FUNCTION_BLOCK FB_Auto_Combination
VAR_INPUT
	bEnable					: BOOL;
END_VAR
VAR_OUTPUT
	fPCV					: LREAL;
	fSCV					: LREAL;
END_VAR
VAR

//Sine Wave
fbClock						: FB_Clock;	
fSineRef					: LREAL;

//Off
fPCV_Off					: LREAL;
fSCV_Off					: LREAL;


//////Primary Control////////
fSCV_On						: LREAL;
fPCV_PC						: LREAL;
	
fbAutoSineMotion_PC			: FB_AutoSineMotion;

/////Secondary Control/////
fPCV_set					: LREAL := 1.0;
fPCV_On						: LREAL;
fSCV_SC						: LREAL;

fbGain_Chooser_P			: FB_GainChooser;
fbGain_Chooser_I			: FB_GainChooser;
fbDerivator					: FB_Derivator;

fbPID_OL					: FB_PID_Controller;
fbDeadband_sine				: FB_Deadband_Auto_sine;
fbDisplacementControl_IL	: FB_DisplacementControl_SC;



//Plotting
fVelref_sine				: LREAL;
fOutPutSignal_OL_combi		: LREAL;
fDeadbandComp_out			: LREAL;

//MUX
fbMUX_selector				: FB_MUX_selector;

END_VAR
VAR // added by the converter: edge detectors and wires of the graphical bodies
    _w1 : LREAL;
    _w2 : BOOL;
END_VAR

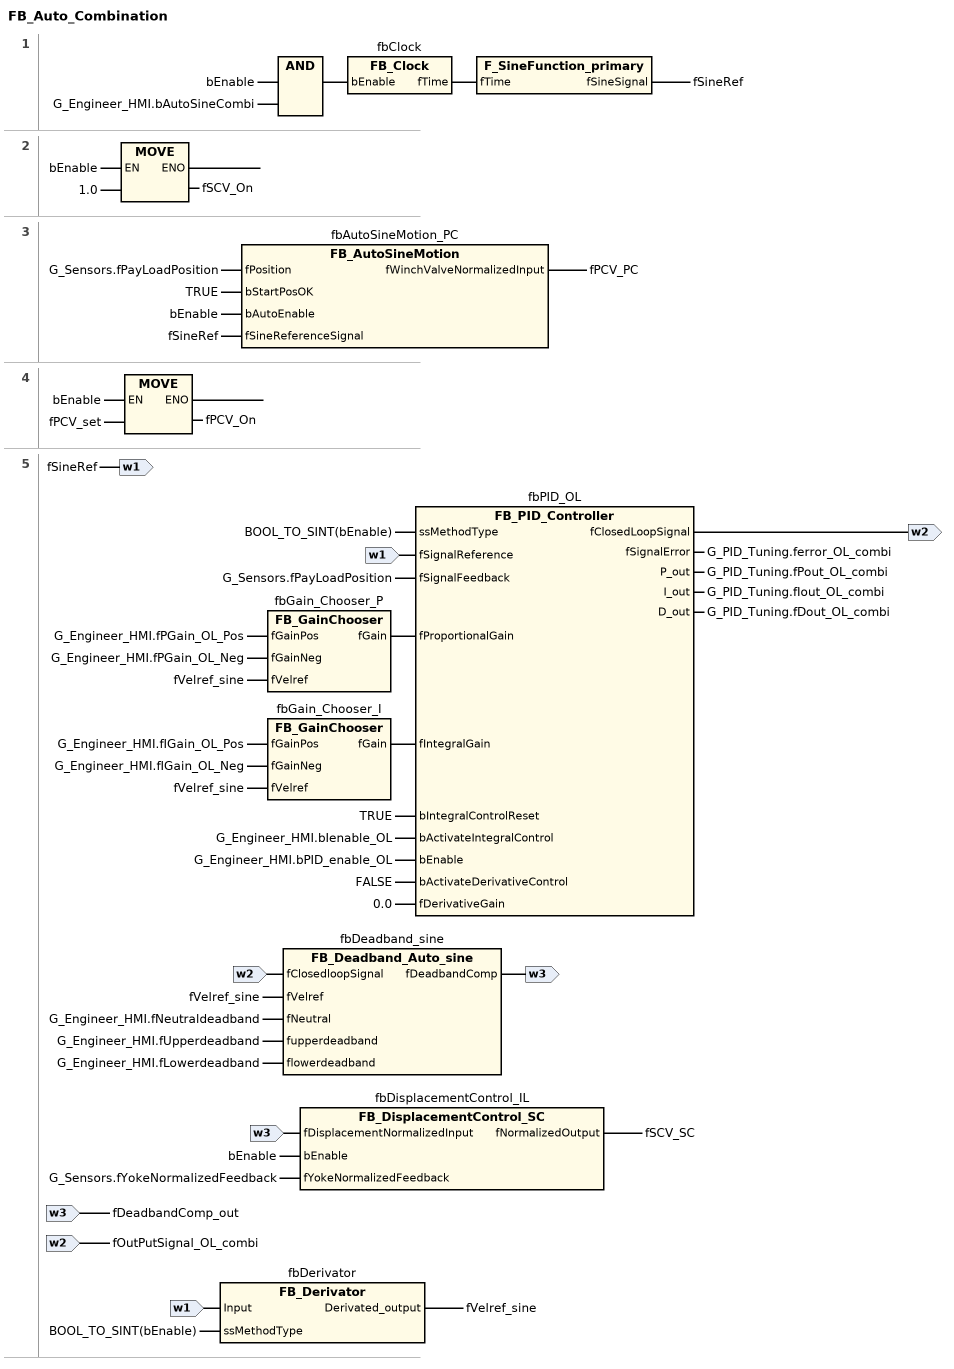
// NETWORK 1
fbClock(bEnable := bEnable AND G_Engineer_HMI.bAutoSineCombi); // FB_Clock
F_SineFunction_primary(fTime := fbClock.fTime, fSineSignal => _w1);
fSineRef := _w1;

// NETWORK 2
IF bEnable THEN fSCV_On := 1.0; END_IF

// NETWORK 3
fbAutoSineMotion_PC(
    fPosition := G_Sensors.fPayLoadPosition,
    bStartPosOK := TRUE,
    bAutoEnable := bEnable,
    fSineReferenceSignal := fSineRef); // FB_AutoSineMotion
fPCV_PC := fbAutoSineMotion_PC.fWinchValveNormalizedInput;

// NETWORK 4
IF bEnable THEN fPCV_On := fPCV_set; END_IF

// NETWORK 5
fbGain_Chooser_P(
    fGainPos := G_Engineer_HMI.fPGain_OL_Pos,
    fGainNeg := G_Engineer_HMI.fPGain_OL_Neg,
    fVelref := fVelref_sine); // FB_GainChooser
fbGain_Chooser_I(
    fGainPos := G_Engineer_HMI.fIGain_OL_Pos,
    fGainNeg := G_Engineer_HMI.fIGain_OL_Neg,
    fVelref := fVelref_sine); // FB_GainChooser
fbPID_OL(
    ssMethodType := BOOL_TO_SINT(bEnable),
    fSignalReference := fSineRef,
    fSignalFeedback := G_Sensors.fPayLoadPosition,
    fProportionalGain := fbGain_Chooser_P.fGain,
    fIntegralGain := fbGain_Chooser_I.fGain,
    bIntegralControlReset := TRUE,
    bActivateIntegralControl := G_Engineer_HMI.bIenable_OL,
    bEnable := G_Engineer_HMI.bPID_enable_OL,
    bActivateDerivativeControl := FALSE,
    fDerivativeGain := 0.0,
    fSignalError => G_PID_Tuning.ferror_OL_combi,
    P_out => G_PID_Tuning.fPout_OL_combi,
    I_out => G_PID_Tuning.fIout_OL_combi,
    D_out => G_PID_Tuning.fDout_OL_combi); // FB_PID_Controller
fbDeadband_sine(
    fClosedloopSignal := fbPID_OL.fClosedLoopSignal,
    fVelref := fVelref_sine,
    fNeutral := G_Engineer_HMI.fNeutraldeadband,
    fupperdeadband := G_Engineer_HMI.fUpperdeadband,
    flowerdeadband := G_Engineer_HMI.fLowerdeadband); // FB_Deadband_Auto_sine
fbDisplacementControl_IL(
    fDisplacementNormalizedInput := fbDeadband_sine.fDeadbandComp,
    bEnable := bEnable,
    fYokeNormalizedFeedback := G_Sensors.fYokeNormalizedFeedback); // FB_DisplacementControl_SC
fSCV_SC := fbDisplacementControl_IL.fNormalizedOutput;
fDeadbandComp_out := fbDeadband_sine.fDeadbandComp;
fOutPutSignal_OL_combi := fbPID_OL.fClosedLoopSignal;
fbDerivator(Input := fSineRef, ssMethodType := BOOL_TO_SINT(bEnable)); // FB_Derivator
fVelref_sine := fbDerivator.Derivated_output;

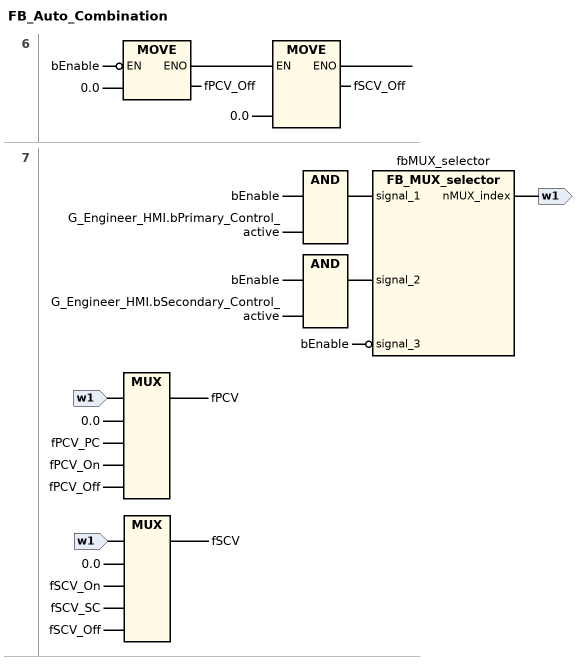
// NETWORK 6
_w2 := NOT bEnable;
IF _w2 THEN fPCV_Off := 0.0; END_IF
IF _w2 THEN fSCV_Off := 0.0; END_IF

// NETWORK 7
fbMUX_selector(
    signal_1 := bEnable AND G_Engineer_HMI.bPrimary_Control_active,
    signal_2 := bEnable AND G_Engineer_HMI.bSecondary_Control_active,
    signal_3 := NOT bEnable); // FB_MUX_selector
fPCV := MUX(fbMUX_selector.nMUX_index, 0.0, fPCV_PC, fPCV_On, fPCV_Off);
fSCV := MUX(fbMUX_selector.nMUX_index, 0.0, fSCV_On, fSCV_SC, fSCV_Off);

END_FUNCTION_BLOCK

(* stored: Version 1.1.0.1
   POU FB_Auto_Combination: Id {26a38f6a-31eb-4cd0-aadd-bbbaf7f3bea7}, SpecialFunc None *)
